Fanuc KAREL source: kt00520.KL

-- PROVISIONAL review KL for V1013-1; original PC SHA256 d9c75bbf1dc41e686586f5ec23c93e45e240d5aabaa1c3cbbc42de3708f9ae06
-- Incomplete behavior may be omitted. Consult companion uncertainty JSON. Do not deploy.
PROGRAM KT00520
%NOLOCKGROUP
-- UNRESOLVED_DECL P1 type=000106
-- UNRESOLVED_DECL P2 type=000102
-- UNRESOLVED_DECL OUT type=000102
BEGIN
  -- UNRESOLVED_PC offsets 5-20; opcodes 2E,22,32,35
  -- UNRESOLVED_PC offsets 25-40; opcodes 2E,22,32,35
  -- UNRESOLVED_PC offsets 45-84; opcodes 49,7E,49,7E,60,7E,4A
  -- UNRESOLVED_PC offsets 89-93; opcodes 7F
END KT00520
